// TwinCAT 3 PLC project Standard
// ProgramVersion: 3.1.4023.0
// libraries:
//   Tc2_Standard, * (Beckhoff Automation GmbH)
//   Tc2_System, * (Beckhoff Automation GmbH)
//   Tc2_Utilities, * (Beckhoff Automation GmbH)
//   Tc3_Module, * (Beckhoff Automation GmbH)
//   Tc3_PLCopen_OpcUa, * (Beckhoff Automation GmbH)
//   Tc2_ModbusSrv,3.3.2.0,Beckhoff Automation GmbH
// project tree:
//   DUTs/ E_EventType.TcDUT, ST_Event.TcDUT
//   / PlcTask.TcTTO
//   POUs/ FB_EventBuffer.TcPOU, FB_ModbusTCPIP_ReadCoils.TcPOU, MAIN.TcPOU
// real-time tasks:
//   TASK PlcTask: cycle T#10ms, priority 20, ADS port 350

CONFIGURATION Standard
    RESOURCE PLC ON TwinCAT3
        TASK PlcTask(INTERVAL := T#10ms, PRIORITY := 20);
        PROGRAM MAIN WITH PlcTask : MAIN;
    END_RESOURCE
END_CONFIGURATION

// ---- DUTs/E_EventType.TcDUT

TYPE E_EventType :
(
	Alarm:= 0,
	Message:= 1,
	Warning:=2
);
END_TYPE

// ---- DUTs/ST_Event.TcDUT
TYPE ST_Event :
STRUCT
	eEventType : E_EventType;
	eEventSeverity : TcEventSeverity;
	nEventIdentity : UDINT;
	nEventText : STRING(255);
	dtTimestamp : DATE_AND_TIME;
END_STRUCT
END_TYPE

// ---- POUs/MAIN.TcPOU
PROGRAM MAIN
VAR
	fbTon : TON := (PT :=T#10S);
	fbTonIN  : BOOL ;
	fbToff : TOF := (PT := T#10S);
	
	fbTrigger : R_TRIG;
	fbTriggerEnable: BOOL;
	upCounter : ULINT;
	
	EventBuffer : FB_EventBuffer;
	
	AddEvent : BOOL;
	stEventToAdd : ST_Event;
	bEventToAddError : BOOL;
	

	
	
	
	GetAndRemoveEvent : BOOL;
	stLastReadEvent  : ST_Event;
	bGetAndRemoveEventError : BOOL;
	
	
	ReadCoilsExample : FB_ModbusTCPIP_ReadCoils;
END_VAR

// Start Main Rutine

fbTon(IN := fbTonIN);
fbToff(IN := fbTonIN);

fbTrigger(CLK := fbTriggerEnable);
IF fbTrigger.Q THEN
	upCounter := upCounter + 1;
END_IF

IF AddEvent THEN
	EventBuffer.AddEvent(stEvent := stEventToAdd, bError => bEventToAddError);
	AddEvent := FALSE;
	END_IF

IF GetAndRemoveEvent THEN
	EventBuffer.GetAndRemoveEvent(stEvent => stLastReadEvent, bError => bGetAndRemoveEventError);
	GetAndRemoveEvent := FALSE;
	
END_IF

ReadCoilsExample();

END_PROGRAM

// ---- POUs/FB_EventBuffer.TcPOU
FUNCTION_BLOCK FB_EventBuffer

VAR
	MemRingBuffer : FB_MemRingBuffer;
	BufferArray : ARRAY[0..NUMBER_OF_BITES_FOR_ALL_ST_EVENT] OF BYTE;
END_VAR

VAR CONSTANT
	SIZE_OF_EVENT : UDINT := SIZEOF(ST_Event);
	MAX_NUMBER_OF_ST_EVENTS : UDINT := 5;
	NUMBER_OF_BITES_FOR_ALL_ST_EVENT : UDINT := SIZE_OF_EVENT * MAX_NUMBER_OF_ST_EVENTS;

END_VAR

METHOD PUBLIC AddEvent
VAR_INPUT
	stEvent : REFERENCE TO ST_Event;
END_VAR
VAR_OUTPUT
	bError : BOOL;
END_VAR
MemRingBuffer.A_AddTail(pWrite := ADR(stEvent),
			            cbWrite := SIZEOF(stEvent),
						pBuffer := ADR(BufferArray),
						cbBuffer := SIZEOF(BufferArray));
bError := NOT MemRingBuffer.bOk;
END_METHOD

METHOD GetAndRemoveEvent
VAR_OUTPUT
	stEvent : ST_Event;
	bError : BOOL;	
END_VAR
MemRingBuffer.A_RemoveHead(pRead := ADR(stEvent),
			            cbRead := SIZEOF(stEvent),
						pBuffer := ADR(BufferArray),
						cbBuffer := SIZEOF(BufferArray));
bError := NOT MemRingBuffer.bOk;
END_METHOD

END_FUNCTION_BLOCK

// ---- POUs/FB_ModbusTCPIP_ReadCoils.TcPOU
FUNCTION_BLOCK FB_ModbusTCPIP_ReadCoils

VAR

fbMBReadCoils : FB_MBReadCoils ;
nReadValue : BYTE;

eReadState : (WAIT, TRIGGER,READ);
fbTrigger : R_TRIG;
END_VAR

fbTrigger();
IF fbTrigger.Q THEN
	IF eReadState = WAIT THEN 
	eReadState := TRIGGER;
	END_IF
END_IF


CASE eReadState OF
	
	WAIT :
	
	// Do nothing
	
	
	TRIGGER :
	
		fbMBReadCoils(
		
		sIPAddr   := '192.168.1.175',
		nTCPPort  := 502,
		nUnitID   := 16#FF,
		nQuantity := 1,
		nMBAddr   := 0,
		cbLength  := SIZEOF(nReadValue),
		pDestAddr := ADR(nReadValue),
		bExecute  := TRUE,
		tTimeout  :=T#5S,
		bBusy=>,
		bError=>,
		nErrId=>,
		cbRead=>,
						);
		eReadState := READ;
	
	READ :
	
	// Here we will be waiting for the response
		fbMBReadCoils(bExecute := FALSE);
		IF NOT fbMBReadCoils.bBusy OR fbMBReadCoils.bError THEN
			eReadState :=WAIT;
			
		END_IF
		
END_CASE

END_FUNCTION_BLOCK
